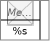
VISUALIZATION VISU_VANNE_2P_H_ACT2  // 50x41
VAR_IN_OUT
	m_Input_VANNE : BLOCK_ACTUATOR2;
END_VAR
    Rectangle (0,0 40x40), invisible if: TRUE
    Polygon (0,0)
    Rectangle (-5,21 50x20), "%s", text variable: m_Input_VANNE.MNEMO
    Polygon (0,0), colour toggle: (m_Input_VANNE.STATE_ON) <> 0, invisible if: NOT (m_Input_VANNE.STATE_OFF OR m_Input_VANNE.STATE_ON)
    Image (7,0 26x25), invisible if: NOT m_Input_VANNE.STATE_Nok, image: MesImages.warning
    Rectangle (0,0 40x20), invisible if: NOT (m_Input_VANNE.Autor_ON_IHM OR m_Input_VANNE.Autor_OFF_IHM) OR NOT PRG_User.ACTU_USER.MAINTENANCE
        tap m_Input_VANNE.M_ON
END_VISUALIZATION

(* stored: Version 1.1.0.1, ProductVersion 3.1.4024.12
   Visu VISU_VANNE_2P_H_ACT2: Id {2937dcbe-326c-4a1c-a8bf-b7ba0bdd5e6d} *)
